PROGRAM Main_T1ms
VAR
			 
END_VAR

// time stamp generation
TimeStamp();

END_PROGRAM

(* stored: Version 1.1.0.1, ProductVersion 3.1.4024.15
   POU Main_T1ms: Id {f7339b70-7acd-4fbe-83cc-3fa441c021ee}, SpecialFunc None *)
